// TIA Portal V19 export
TYPE "UDT_SIM_VLV"
   STRUCT
      simMain : Bool;
      simUpper : Bool;
      simLower : Bool;
      simDeact : Bool;
   END_STRUCT;
END_TYPE
